# EPICS substitutions: db/Beckhoff_4XXX/ecmcEL4374.substitutions
file "ecmc_analogInput-chX.template"
{
  pattern {CH_ID, ESLO, EOFF, EGU, PREC, LOW, LOLO, HIGH, HIHI, HYST, LLSV, LSV, HSV, HHSV}
          {01, "${_ESLO=1}", "${_EOFF=0}", "${_EGU=Raw}", "${_PREC=0}", -32768, -32769, 32769, 32770, 0, "MAJOR", "MINOR", "MINOR", "MAJOR"}
          {02, "${_ESLO=1}", "${_EOFF=0}", "${_EGU=Raw}", "${_PREC=0}", -32768, -32769, 32769, 32770, 0, "MAJOR", "MINOR", "MINOR", "MAJOR"}
}

file "ecmc_status_analog-chX.template"
{
  pattern {CH_ID, KEY }
          {01,    "AI"}
          {02,    "AI"}
}

file "ecmc_analogOutput-chX.template"
{
  pattern {CH_ID, ESLO, EOFF, EGU, PREC, LOW, LOLO, HIGH, HIHI, HYST, LLSV, LSV, HSV, HHSV, DRVL, DRVH}
          {01, "${_ESLO=1}", "${_EOFF=0}", "${_EGU=Raw}", "${_PREC=0}", -32768, -32769, 32769, 32770, 0, "MAJOR", "MINOR", "MINOR", "MAJOR", -32767, 32768}
          {02, "${_ESLO=1}", "${_EOFF=0}", "${_EGU=Raw}", "${_PREC=0}", -32768, -32769, 32769, 32770, 0, "MAJOR", "MINOR", "MINOR", "MAJOR", -32767, 32768}
}
